# EPICS substitutions: db/Beckhoff_5XXX/ecmcEL5001.substitutions
file "ecmcEcSlave.template"
{
  pattern {}
          {}
}

file "ecmcEL5001-chX.template"
{
  pattern {LINR,    ESLO,   EOFF,   EGU,        PREC, LOW, LOLO, HIGH, HIHI, HYST, LLSV,       LSV,        HSV,        HHSV      }
          {"SLOPE", 1,      0,      "Steps",    0,    0,   0,    0,    0,    0,    "NO_ALARM", "NO_ALARM", "NO_ALARM", "NO_ALARM"}
}
